// TIA Portal V17 export
// export: Created 2023-12-22T15:05:29.8399383Z, ExportSetting WithDefaults, DisplayName Totally Integrated Automation Portal, DisplayVersion V17, DisplayName TIA Portal Openness, DisplayVersion V17, DisplayName TIA Portal Version Control Interface, DisplayVersion V17, DisplayName STEP 7 Professional, DisplayVersion V17, DisplayName STEP 7 Safety, DisplayVersion V17, DisplayName WinCC Advanced, DisplayVersion V17
DATA_BLOCK "DIx_1_DB"   // DB200
VERSION : 0.1
// stored: AutoNumber false, DBAccessibleFromOPCUA true, InstanceOfName DIx_1, InstanceOfType FB
"DIx_1"
   // VAR RETAIN
   //    AllBlock { S7_SetPoint := 'True'} : "DI_ex";
   //    EZ_1_FB_AHLS { S7_SetPoint := 'True'} : "DI_ex";
   //    Gas_Chanel_1_1 { S7_SetPoint := 'True'} : "DI_ex";
   //    Gas_Chanel_1_2 { S7_SetPoint := 'True'} : "DI_ex";
   //    Gas_Chanel_2_1 { S7_SetPoint := 'True'} : "DI_ex";
   //    Gas_Chanel_2_2 { S7_SetPoint := 'True'} : "DI_ex";
   //    ALS_1 { S7_SetPoint := 'True'} : "DI_ex";
   //    KC_1 { S7_SetPoint := 'True'} : "DI_ex";
   //    KC_2 { S7_SetPoint := 'True'} : "DI_ex";
   //    signal_10 { S7_SetPoint := 'True'} : "DI_ex";
   //    signal_11 { S7_SetPoint := 'True'} : "DI_ex";
   //    signal_12 { S7_SetPoint := 'True'} : "DI_ex";
   //    signal_13 { S7_SetPoint := 'True'} : "DI_ex";
   //    Time_DTL { S7_SetPoint := 'True'} : DTL := DTL#2012-01-01-20:29:24.070589;
   // END_VAR
BEGIN
   AllBlock.Use.Inverse := TRUE;
   AllBlock.Use.Indirect := TRUE;
   AllBlock.ADDR_Byte := 1;
   AllBlock.ADDR_Bit := 5;
   AllBlock.Filter_On.SP := 16#02;
   AllBlock.Filter_Off.SP := 16#02;
   EZ_1_FB_AHLS.Use.Inverse := TRUE;
   EZ_1_FB_AHLS.Use.Indirect := TRUE;
   EZ_1_FB_AHLS.ADDR_Byte := 2;
   EZ_1_FB_AHLS.ADDR_Bit := 2;
   EZ_1_FB_AHLS.Filter_On.SP := 16#02;
   EZ_1_FB_AHLS.Filter_Off.SP := 16#02;
   Gas_Chanel_1_1.Use.Inverse := TRUE;
   Gas_Chanel_1_1.Use.Indirect := TRUE;
   Gas_Chanel_1_1.ADDR_Byte := 0;
   Gas_Chanel_1_1.ADDR_Bit := 7;
   Gas_Chanel_1_1.Filter_On.SP := 16#02;
   Gas_Chanel_1_1.Filter_Off.SP := 16#02;
   Gas_Chanel_1_2.Use.Inverse := TRUE;
   Gas_Chanel_1_2.Use.Indirect := TRUE;
   Gas_Chanel_1_2.ADDR_Byte := 1;
   Gas_Chanel_1_2.ADDR_Bit := 0;
   Gas_Chanel_1_2.Filter_On.SP := 16#02;
   Gas_Chanel_1_2.Filter_Off.SP := 16#02;
   Gas_Chanel_2_1.Use.Inverse := TRUE;
   Gas_Chanel_2_1.Use.Indirect := TRUE;
   Gas_Chanel_2_1.ADDR_Byte := 1;
   Gas_Chanel_2_1.ADDR_Bit := 1;
   Gas_Chanel_2_1.Filter_On.SP := 16#02;
   Gas_Chanel_2_1.Filter_Off.SP := 16#02;
   Gas_Chanel_2_2.Use.Inverse := TRUE;
   Gas_Chanel_2_2.Use.Indirect := TRUE;
   Gas_Chanel_2_2.ADDR_Byte := 1;
   Gas_Chanel_2_2.ADDR_Bit := 2;
   Gas_Chanel_2_2.Filter_On.SP := 16#02;
   Gas_Chanel_2_2.Filter_Off.SP := 16#02;
   ALS_1.Use.Inverse := FALSE;
   ALS_1.Use.Indirect := TRUE;
   ALS_1.ADDR_Byte := 2;
   ALS_1.ADDR_Bit := 0;
   ALS_1.Filter_On.SP := 16#02;
   ALS_1.Filter_Off.SP := 16#02;
   KC_1.Use.Inverse := FALSE;
   KC_1.Use.Indirect := TRUE;
   KC_1.ADDR_Byte := 1;
   KC_1.ADDR_Bit := 3;
   KC_1.Filter_On.SP := 16#02;
   KC_1.Filter_Off.SP := 16#02;
   KC_2.Use.Inverse := FALSE;
   KC_2.Use.Indirect := TRUE;
   KC_2.ADDR_Byte := 1;
   KC_2.ADDR_Bit := 4;
   KC_2.Filter_On.SP := 16#02;
   KC_2.Filter_Off.SP := 16#02;
   signal_10.Use.Inverse := TRUE;
   signal_10.Use.Indirect := TRUE;
   signal_10.ADDR_Byte := 2;
   signal_10.ADDR_Bit := 7;
   signal_10.Filter_On.SP := 16#02;
   signal_10.Filter_Off.SP := 16#02;
   signal_11.Use.Inverse := TRUE;
   signal_11.Use.Indirect := TRUE;
   signal_11.ADDR_Byte := 2;
   signal_11.ADDR_Bit := 5;
   signal_11.Filter_On.SP := 16#02;
   signal_11.Filter_Off.SP := 16#02;
   signal_12.Use.Inverse := TRUE;
   signal_12.Use.Indirect := TRUE;
   signal_12.ADDR_Byte := 2;
   signal_12.ADDR_Bit := 6;
   signal_12.Filter_On.SP := 16#02;
   signal_12.Filter_Off.SP := 16#02;
   signal_13.Use.Inverse := TRUE;
   signal_13.Use.Indirect := TRUE;
   signal_13.ADDR_Byte := 3;
   signal_13.ADDR_Bit := 0;
   signal_13.Filter_On.SP := 16#02;
   signal_13.Filter_Off.SP := 16#02;
END_DATA_BLOCK
